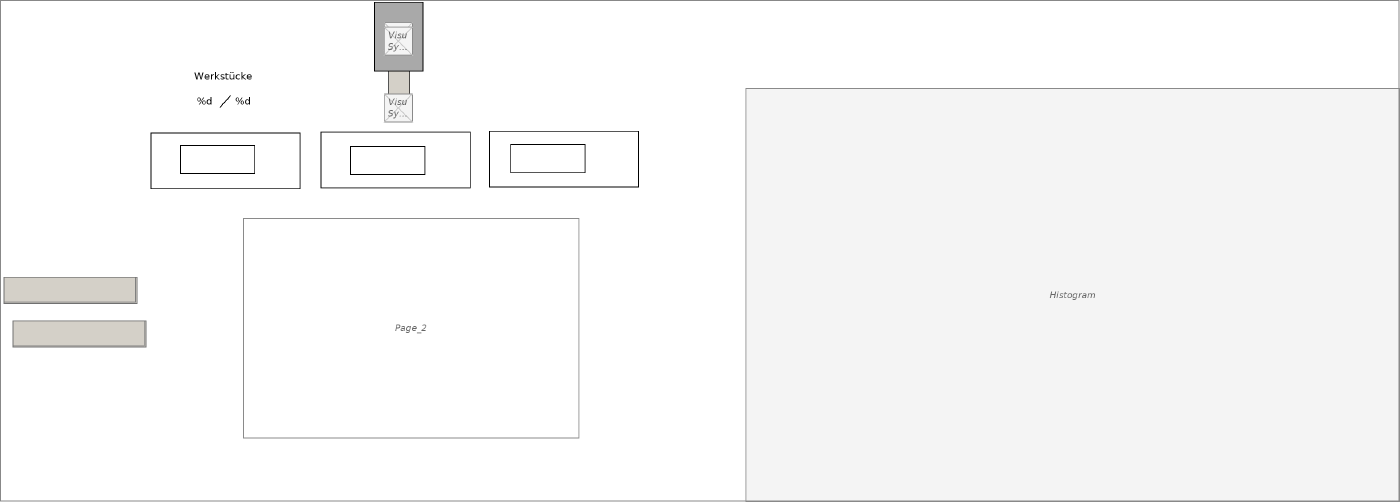
VISUALIZATION Visualization  // 1572x564
    RoundedRectangle (169,149 168x63), colour toggle: GVL_HMI.Status_Band_3, colour variable: 16#ff999999
        p3450524324: 16#00555555
        p2167032090: 16#ff00FF00
        p3092690914: 16#00555555
    RoundedRectangle (360,148 168x63), colour toggle: GVL_HMI.Status_Band_2, colour variable: 16#ff999999
        p3450524324: 16#00555555
        p2167032090: 16#ff00FF00
        p3092690914: 16#00555555
    RoundedRectangle (549,147 168x63), colour toggle: GVL_IO.A_Band_1, colour variable: 16#ff999999
        p2167032090: 16#ff00FF00
        p3450524324: 16#00555555
        p3092690914: 16#00555555
    RoundedRectangle (573,162 84x32), colour toggle: GVL_IO.E_LT_Band_1, colour variable: 16#00555555
        p2167032090: 16#ffc3863c
        p3450524324: 16#00555555
        p3092690914: 16#00555555
    RoundedRectangle (393,164 84x32), colour toggle: GVL_IO.E_LT_Band_2, colour variable: 16#00555555
        p2167032090: 16#ffc3863c
        p3450524324: 16#00555555
        p3092690914: 16#00555555
    RoundedRectangle (202,163 84x32), colour toggle: GVL_IO.E_LT_Band_3, colour variable: 16#00555555
        p2167032090: 16#ffc3863c
        p3450524324: 16#00555555
        p3092690914: 16#00555555
    RoundedRectangle (436,76 24x51)
    RoundedRectangle (420,2 55x78)
    Image (431,105 32x32), invisible if: GVL_HMI.Status_Bohrer_inv, image: VisuSymbols.Symbols.ArrowHalfRightDown
    Image (431,25 32x32), colour toggle: GVL_IO.A_Bohrwerk_zurueck, invisible if: GVL_HMI.Status_BW_Zur_inv, image: VisuSymbols.Symbols.ArrowBoldUp
        p573394764: 16#FF00FF00
        p2175578022: 16#FF000000
    Image (431,30 32x32), invisible if: GVL_HMI.Status_BW_Vor_inv, image: VisuSymbols.Symbols.ArrowBoldDown
    Group (209,71 84x58)
        Label (0,0 84x30), "Werkstücke"
        Rectangle (3,28 36x30), "%d", text variable: PRG_MAIN.fb_Antriebe.FB_Automatik_inst.CTU_Werkstueckzaehler.CV
        Rectangle (47,28 34x30), "%d", text variable: PRG_MAIN.fb_Antriebe.FB_Automatik_inst.CTU_Werkstueckzaehler.PV
        Line (38,49) (50,36)
    Histogram (837,99 735x465), scale format: %.1f, scale 0..100
        p518627256: mm
        p1518820177: GVL_GlobalData.DataArray
        p102497268: GVL_GlobalData.DataArray
        p788070771: ARRAY [0..100] OF DINT
    Button (4,311 150x30)
    Button (14,360 150x30)
    Frame (273,245 377x247)
        shows Page_2()
END_VISUALIZATION

(* stored: Version 1.1.0.1, ProductVersion 3.1.4024.12
   Visu Visualization: Id {5c285192-c964-4a1a-8145-1a0392c00098} *)
